Universal Robots PolyScope program: Ejercicio_3.urp

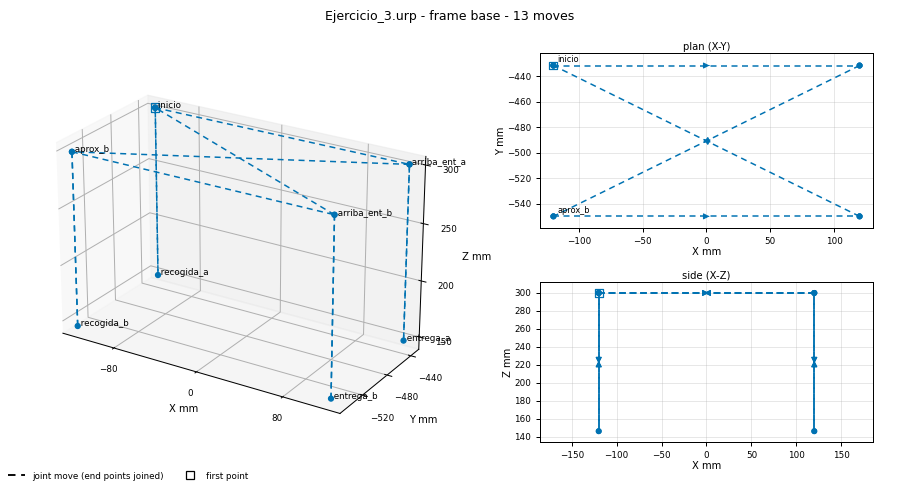
[picture p0: tool path of Ejercicio_3.urp in frame base, 13 of 13 moves have a stored position in this frame; points joined in program order, loops and branches not executed]
Program Ejercicio_3 (installation=default directory=/ursim/programs createdIn=3.15.8.106339 lastSavedIn=3.15.8.106339 robotSerialNumber=2018359999)
Calibrated DH parameters: a=[0, -0.425, -0.39225, 0, 0, 0]; d=[0.089159, 0, 0, 0.10915, 0.09465, 0.0823]; alpha=[1.570796, 0, 0, 1.570796, -1.570796, 0]; deltaTheta=[0, 0, 0, 0, 0, 0]
Robot Program (runOnlyOnce=false)
  MoveJ speed 30 deg/s, acceleration 60 deg/s^2 (useActiveTCP=true)
    Set DigitalOutput (payload=0.5 tcpAsCog=true) pin=digital_out[0]; digitalValue=0
    Waypoint inicio: TCP in base x=-120 y=-431.763 z=300 mm, rx=-0.0012 ry=3.1163 rz=0.0389 rad; joints [-91.699, -86.228, -112.904, -72.341, 91.393, -1.761] deg
    Waypoint recogida_a: TCP in base x=-120 y=-431.763 z=146.07 mm, rx=-0.0012 ry=3.1163 rz=0.0389 rad; joints [-91.699, -98.952, -126.227, -46.293, 91.393, -1.761] deg
    Set DigitalOutput (payload=1 tcpAsCog=true) pin=digital_out[0]; digitalValue=1
    Wait Sleep waitTime=0.5
    Waypoint arriba_a: TCP in base x=-120 y=-431.763 z=300 mm, rx=-0.0012 ry=3.1163 rz=0.0389 rad; joints [-91.699, -86.228, -112.904, -72.341, 91.393, -1.761] deg
    Waypoint arriba_ent_a: TCP in base x=120 y=-431.763 z=300 mm, rx=-0.0012 ry=3.1163 rz=0.0389 rad; joints [-60.74, -86.141, -113.221, -71.184, 91.952, 29.206] deg
    Waypoint entrega_a: TCP in base x=120 y=-431.763 z=146.07 mm, rx=-0.0012 ry=3.1163 rz=0.0389 rad; joints [-60.74, -98.998, -126.489, -45.06, 91.952, 29.206] deg
    Set DigitalOutput (payload=0.5 tcpAsCog=true) pin=digital_out[0]; digitalValue=0
    Wait Sleep waitTime=0.5
    Waypoint salida_a: TCP in base x=120 y=-431.763 z=300 mm, rx=-0.0012 ry=3.1163 rz=0.0389 rad; joints [-60.74, -86.141, -113.221, -71.184, 91.952, 29.206] deg
    Waypoint aprox_b: TCP in base x=-120 y=-550 z=300 mm, rx=-0.0012 ry=3.1163 rz=0.0389 rad; joints [-91.337, -101.793, -96.101, -73.57, 91.402, -1.4] deg
    Waypoint recogida_b: TCP in base x=-120 y=-550 z=146.07 mm, rx=-0.0012 ry=3.1163 rz=0.0389 rad; joints [-91.337, -112.079, -107.944, -51.441, 91.402, -1.4] deg
    Set DigitalOutput (payload=1 tcpAsCog=true) pin=digital_out[0]; digitalValue=1
    Wait Sleep waitTime=0.5
    Waypoint arriba_b: TCP in base x=-120 y=-550 z=300 mm, rx=-0.0012 ry=3.1163 rz=0.0389 rad; joints [-91.337, -101.793, -96.101, -73.57, 91.402, -1.4] deg
    Waypoint arriba_ent_b: TCP in base x=120 y=-550 z=300 mm, rx=-0.0012 ry=3.1163 rz=0.0389 rad; joints [-66.792, -101.724, -96.367, -72.658, 91.884, 23.15] deg
    Waypoint entrega_b: TCP in base x=120 y=-550 z=146.07 mm, rx=-0.0012 ry=3.1163 rz=0.0389 rad; joints [-66.792, -112.088, -108.156, -50.505, 91.884, 23.15] deg
    Set DigitalOutput (payload=0.5 tcpAsCog=true) pin=digital_out[0]; digitalValue=0
    Waypoint salida_b: TCP in base x=120 y=-550 z=300 mm, rx=-0.0012 ry=3.1163 rz=0.0389 rad; joints [-66.792, -101.724, -96.367, -72.658, 91.884, 23.15] deg
    Waypoint Waypoint_2: TCP in base x=-120 y=-431.76 z=300 mm, rx=-0.0012 ry=3.1163 rz=0.0389 rad; joints [-91.699, -86.228, -112.904, -72.341, 91.393, -1.761] deg
    Wait DigitalInput pin=digital_in[0]; digitalValue=0
    Wait DigitalInput pin=digital_in[0]; digitalValue=1
